TYPE UDT_Crimping_RD :
STRUCT
  
Imm : UDT_Imm_Crimping_RD;
Message : UDT_StationMessage_RD;
Hmi : UDT_Hmi_Crimping_RD;

UnitState : INT;	//DISABLED := 1,OPERATIONAL :=2,STANDBY :=3,UNKNOWN :=4
Command :INT; //INIT :=1,START := 2,STOP :=3,PAUSE := 4
CommandState : INT ; 	//NOT_READY := 1,READY :=2,RUNNING :=3,DONE :=4,CANCEL :=5,INIT := 6,ERROR :=7

END_STRUCT
END_TYPE

(* stored: Version 1.1.0.1, ProductVersion 3.1.4024.12
   DUT UDT_Crimping_RD: Id {ed3dd117-0c47-44b8-a36a-97ba8fefc3eb} *)
